TYPE TYP_HW_EL6001_OUT :
STRUCT
	COM AT %Q* : KL6OutData22B;
END_STRUCT
END_TYPE

(* stored: Version 1.1.0.1, ProductVersion 3.1.4024.12
   DUT TYP_HW_EL6001_OUT: Id {1afbba61-05bd-4e2c-8111-0c415e301542} *)
